(*
SPDX-FileCopyrightText: © 2026 Oleksandr Tiutyk <trofimich@gmail.com>
SPDX-License-Identifier: MIT
License: https://opensource.org/license/mit
*)

INTERFACE IAggregateException EXTENDS IException

METHOD GetInnerException : IException
VAR_INPUT
	index : DINT;
END_VAR
END_METHOD

METHOD GetRootException : IException
END_METHOD

{attribute 'monitoring' := 'call'}
PROPERTY InnerExceptionCount : UINT
GET
END_GET
END_PROPERTY

METHOD Throw
VAR_INPUT
	sourceNamespaceName : STRING;
	sourceClassName : STRING;
	sourcePOUName : STRING;
	sourcePosition : STRING;
END_VAR
END_METHOD

END_INTERFACE

(* stored: Version 1.1.0.1
   Itf IAggregateException: Id {b988b248-0471-4475-9d2a-afe0ffc9eec0}
   Method GetInnerException: Id {2d916ec4-46b0-4973-8bf3-5e92184d2ef7}
   Method GetRootException: Id {05287103-fa2a-4150-b3ca-bf42a00677a5}
   Property InnerExceptionCount: Id {667bfa13-f04a-4a29-8276-1126128becce}
   Get Get: Id {730d4a93-a9ce-44b8-a0bd-f31516351203}
   Method Throw: Id {c37a3a93-2628-4dc7-9856-dab793c214a9} *)
